FUNCTION_BLOCK PUBLIC MoveMoverToPositionZoned EXTENDS MoveMoverToPosition
VAR_INPUT
END_VAR
VAR_OUTPUT
END_VAR
VAR
	i: INT;
	StartZone: INT;
	CurrentZone : INT;
	ZoneTransitionPositions : ARRAY[1..4] OF DINT;
	ZoneVelocities : ARRAY[1..4] OF MC_LREAL;
END_VAR

CASE State OF
	0:
		IF _MoveMover THEN
			_done := FALSE;
			_error := FALSE;
			_busy := TRUE;
			moveAbs.Execute := TRUE;
			StartZone := GetZone();
			moveAbs.Velocity := ZoneVelocities[StartZone];
			IF moveAbs.Busy THEN
				State := 10;
				_MoveMover := FALSE;
			END_IF
		END_IF
	
	10:
		IF NOT moveAbs.Busy THEN
			IF moveAbs.Done THEN
				_done := TRUE;
			ELSIF moveAbs.Error THEN
				_error := TRUE;
			END_IF
			_busy := FALSE;
			moveAbs.Execute := FALSE;
			State := 0;
		ELSE
			CurrentZone := GetZone();
			IF CurrentZone <> StartZone THEN
				moveAbs.Execute := FALSE;
				State := 0;
				_MoveMover := TRUE;
			END_IF
		END_IF
END_CASE

moveAbs(Axis := _axis);

METHOD FB_init : BOOL
VAR_INPUT
	bInitRetains : BOOL; // if TRUE, the retain variables are initialized (warm start / cold start)
	bInCopyCode : BOOL;  // if TRUE, the instance afterwards gets moved into the copy code (online change)
	axis : REFERENCE TO AXIS_REF;
	arrPositions : ARRAY[1..4] OF DINT;
	arrVelos : ARRAY[1..4] OF MC_LREAL;
END_VAR
SUPER^();
ZoneTransitionPositions := arrPositions;
ZoneVelocities := arrVelos;
END_METHOD

METHOD GetZone : int
VAR_INPUT
END_VAR
IF _axis.NcToPlc.ModuloActPos > ZoneTransitionPositions[1] AND _axis.NcToPlc.ModuloActPos < ZoneTransitionPositions[2] THEN
	GetZone := 1;
ELSIF (_axis.NcToPlc.ModuloActPos > ZoneTransitionPositions[2] AND _axis.NcToPlc.ModuloActPos < 11000.0) 
		OR _axis.NcToPlc.ModuloActPos > 0.0 AND  _axis.NcToPlc.ModuloActPos < ZoneTransitionPositions[3] THEN
	GetZone := 2;
ELSIF _axis.NcToPlc.ModuloActPos > ZoneTransitionPositions[3] AND _axis.NcToPlc.ModuloActPos < ZoneTransitionPositions[4] THEN
	GetZone := 3;
ELSIF _axis.NcToPlc.ModuloActPos > ZoneTransitionPositions[4] THEN
	GetZone := 4;
ELSE
	GetZone := 4;
END_IF
END_METHOD

END_FUNCTION_BLOCK

(* stored: Version 1.1.0.1, ProductVersion 3.1.4024.11
   POU MoveMoverToPositionZoned: Id {8bf14309-c05e-4e32-a9cf-c640451f85c6}, SpecialFunc None
   Method FB_init: Id {6ee86efb-83b0-4bbc-9b17-a763f7f90ce4}
   Method GetZone: Id {50824bdc-8788-4c2d-b3ea-cd5268c03d38} *)
